Staubli VAL3: stop.pgx

program stop()
begin
  resetMotion()
  popUpMsg("Pending movement commands have been cancelled.")
  cls()
end
